Staubli VAL3: InitSocket.pgx

public program InitSocket()
  local num l_nSocket
begin
  l_nSocket=clearBuffer(socket)
end
